# B&R Automation Studio project prak4
Automation Studio 4.5.2.102

## Configuration Config1

### Hardware
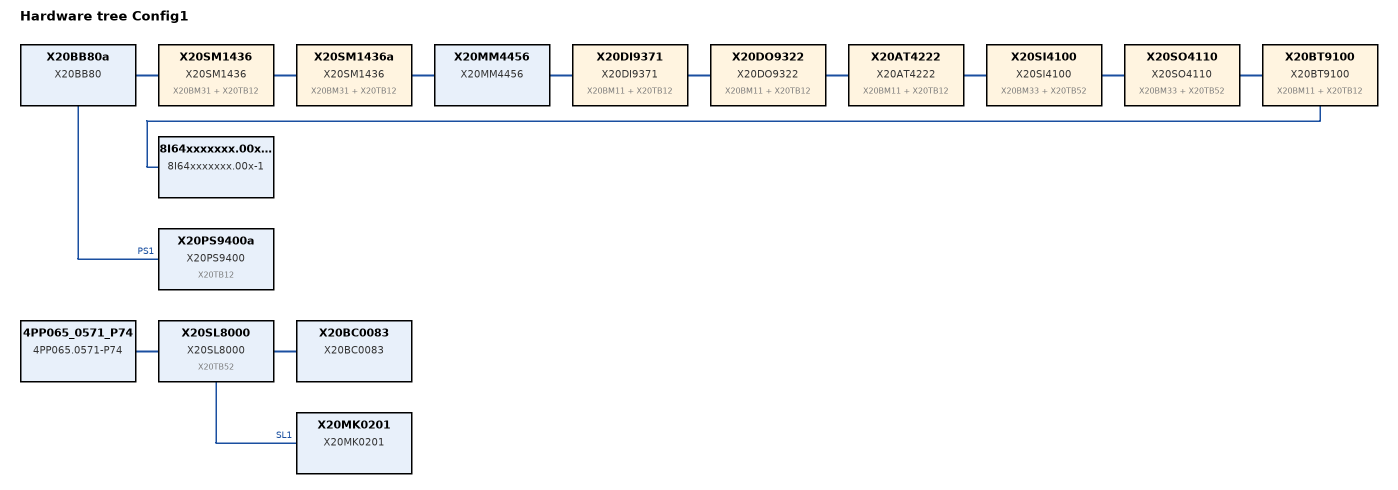
```
4PP065_0571_P74 : 4PP065.0571-P74 v1.1.2.0
  Connector IF5:
    ActivateDevice = 1
    Mode = Manual
    InternetAddress = 10.0.1.10
    SubnetMask = 255.255.255.0
  ConfigurationID = labBR
  TimerDeviceType = EPLX2X
  TimerDevice = 4PP065_0571_P74.IF4
  TaskClassIdleTime = 2000
  Cyclic1Duration = 2000
  Cyclic1Tolerance = 0
  Cyclic1Output = 1
  VcObjectName = Visu
8I64xxxxxxx.00x-1 : 8I64xxxxxxx.00x-1 v2.1.2.0  [X2X1 -> X20BT9100.X2X1 [Cable Type=X2XCable, Length=10, Version=1.0.0.2]]
  packedETAD = packed
  packedCMDD = packed
X20AT4222 : X20AT4222 v1.2.3.0  [SS1 -> X20TB12e.SS; SL -> X20BM11b.SL1]
X20BB80a : X20BB80 v1.0.2.0
X20BC0083 : X20BC0083 v2.9.0.0  [PLK1 -> X20SL8000.PLK2 [Cable Type=PowerlinkCable, Length=10, Version=1.0.0.2]; SL -> X20BB80a.SL1]
X20BM11 : X20BM11 v1.0.0.1  [X2X1 -> X20MM4456.X2X2]
X20BM11a : X20BM11 v1.0.0.1  [X2X1 -> X20BM11.X2X2]
X20BM11b : X20BM11 v1.0.0.1  [X2X1 -> X20BM11a.X2X2]
X20BM11c : X20BM11 v1.0.0.1  [X2X1 -> X20BM33a.X2X2]
X20BM31 : X20BM31 v1.0.0.1  [X2X1 -> X20BB80a.IF1]
X20BM31a : X20BM31 v1.0.0.1  [X2X1 -> X20BM31.X2X2]
X20BM33 : X20BM33 v1.0.0.4  [X2X1 -> X20BM11b.X2X2]
X20BM33a : X20BM33 v1.0.0.4  [X2X1 -> X20BM33.X2X2]
X20BT9100 : X20BT9100 v1.0.3.0  [SS1 -> X20TB12f.SS; SL -> X20BM11c.SL1]
X20DI9371 : X20DI9371 v1.0.2.0  [SS1 -> X20TB12c.SS; SL -> X20BM11.SL1]
X20DO9322 : X20DO9322 v1.0.3.0  [SS1 -> X20TB12d.SS; SL -> X20BM11a.SL1]
X20MK0201 : X20MK0201 v1.0.0.0  [SL -> X20SL8000.SL1]
X20MM4456 : X20MM4456 v1.1.5.0  [X2X1 -> X20BM31a.X2X2]
X20PS9400a : X20PS9400 v1.0.2.4  [SS1 -> X20TB12a.SS; PS -> X20BB80a.PS1]
X20SI4100 : X20SI4100 v1.10.1.1  [SS1 -> X20TB52a.SS; SL -> X20BM33.SL1]
X20SL8000 : X20SL8000 v1.6.5.1  [PLK1 -> 4PP065_0571_P74.IF4 [Cable Type=PowerlinkCable, Length=10, Version=1.0.0.2]; PLK2 -> X20BC0083.PLK1 [Cable Type=PowerlinkCable, Length=10, Version=1.0.0.2]; SS1 -> X20TB52.SS]
  SafeProject = SafeLOGIC-1
X20SM1436 : X20SM1436 v1.4.2.1  [SS1 -> X20TB12.SS; SL -> X20BM31.SL1]
X20SM1436a : X20SM1436 v1.4.2.1  [SS1 -> X20TB12b.SS; SL -> X20BM31a.SL1]
X20SO4110 : X20SO4110 v1.10.1.1  [SS1 -> X20TB52b.SS; SL -> X20BM33a.SL1]
  SafeModuleID = 3
X20TB12 : X20TB12 v1.0.0.0
X20TB12a : X20TB12 v1.0.0.0
X20TB12b : X20TB12 v1.0.0.0
X20TB12c : X20TB12 v1.0.0.0
X20TB12d : X20TB12 v1.0.0.0
X20TB12e : X20TB12 v1.0.0.0
X20TB12f : X20TB12 v1.0.0.0
X20TB52 : X20TB52 v1.0.0.1
X20TB52a : X20TB52 v1.0.0.1
X20TB52b : X20TB52 v1.0.0.1
```

### IoMap.iom - 4PP065_0571_P74/IoMap.iom
```iecst
VAR_CONFIG
	Cyclic#1.gAxis02_DrvIf.iLifeCnt AT %IB."8I64xxxxxxx.00x-1".SDC_LifeCnt;
	Cyclic#1.gAxis02_DrvIf.iDrvOK AT %IX."8I64xxxxxxx.00x-1".ETAD_Input_Bool_02;
	Cyclic#1.gAxis02_DrvIf.oSetTime AT %QW."8I64xxxxxxx.00x-1".SDC_SetTime;
	::Program:speed AT %QW."8I64xxxxxxx.00x-1".LFRD_Output;
	Cyclic#1.gAxis02_DiDoIf.iLifeCntDriveReady AT %IB."8I64xxxxxxx.00x-1".SDC_LifeCnt;
	Cyclic#1.gAxis02_DiDoIf.iLifeCntDriveEnable AT %IB."8I64xxxxxxx.00x-1".SDC_LifeCnt;
	Cyclic#1.gAxis02_DiDoIf.oDriveEnable AT %QX."8I64xxxxxxx.00x-1".CMDD_Output_Bool_00;
	Cyclic#1.gAxis02_ModuleOk AT %QX."8I64xxxxxxx.00x-1".CMDD_Output_Bool_01;
	Cyclic#1.gAxis02_ModuleOk AT %QX."8I64xxxxxxx.00x-1".CMDD_Output_Bool_02;
	Cyclic#1.gAxis02_ModuleOk AT %IX."8I64xxxxxxx.00x-1".ModuleOk;
	Cyclic#1.gAxis02_DiDoIf.oDriveEnable AT %QX."8I64xxxxxxx.00x-1".CMDD_Output_Bool_03;
	Cyclic#1.gAxis02_DiDoIf.iDriveReady AT %IX."8I64xxxxxxx.00x-1".ETAD_Input_Bool_02;
	EVIRD.STATE AT %IW."8I64xxxxxxx.00x-1".ETAD_Input;
	::EVIRD.COM AT %QW."8I64xxxxxxx.00x-1".CMDD_Output;
	::led1 AT %QX."X20DO9322".DigitalOutput02;
	::led2 AT %QX."X20DO9322".DigitalOutput03;
	::led3 AT %QX."X20DO9322".DigitalOutput04;
	::led4 AT %QX."X20DO9322".DigitalOutput05;
	::EVIRD.real_speed AT %IW."8I64xxxxxxx.00x-1".RFRD_Input;
END_VAR
```

### Acp10map.ncm - 4PP065_0571_P74/Motion/Acp10map.ncm
```
NcMapping (NcSwId=Acp10)
  NcObject X20SM1436_ncAXIS1 (ModuleId=X20SM1436, ModuleAddress=SDC_IF1.ST1, Type=ncAXIS, Channel=1, AcoposSimulation=Off, Disabled=TRUE, ModuleDisabled=FALSE)
  NcObject X20SM1436a_ncAXIS1 (ModuleId=X20SM1436a, ModuleAddress=SDC_IF1.ST2, Type=ncAXIS, Channel=1, AcoposSimulation=Off, Disabled=TRUE, ModuleDisabled=FALSE)
  NcObject gAxis02 (ModuleId=8I64xxxxxxx.00x-1, ModuleAddress=SDC_IF1.ST3, Type=ncAXIS, Channel=1, AcoposSimulation=Off, InitParameter=gAxis02i, AcoposParameter=gAxis02a, Disabled=FALSE, ModuleDisabled=FALSE)
```

## Logical view

Binary libraries used (declarations not repeated): operator, runtime, astime, AsIecCon, Acp10man, Acp10par, NcGlobal, Acp10sdc, AsBrStr, Acp10_MC, brsystem, sys_lib

### Global.var - Global variables
```iecst
VAR
	gAxis01 : ACP10AXIS_typ;
	gAxis01_HW : SdcHwCfg_typ := (0);
	gAxis01_DrvIf : SdcDrvIf16_typ := (0);
	gAxis01_DiDoIf : SdcDiDoIf_typ := (0);
	gAxis01_ModuleOk : BOOL := 0;
	gAxis02 : ACP10AXIS_typ;
	gAxis02_HW : SdcHwCfg_typ := (0);
	gAxis02_DrvIf : SdcDrvIf16_typ := (0);
	gAxis02_DiDoIf : SdcDiDoIf_typ := (0);
	gAxis02_ModuleOk : BOOL := 0;
	EVIRD : DRIVE;
	led1 : BOOL;
	led2 : BOOL;
	led3 : BOOL;
	led4 : BOOL;
END_VAR
```

### Package Logical/Libraries - Global libraries

- Visualisation Logical/Libraries/Visu (not shown)

### Program Logical/Program (ANSIC)

#### Variables.var
```iecst
VAR
	speed : INT;
END_VAR
```

#### Main.c
```c
#include <bur/plctypes.h>

#ifdef _DEFAULT_INCLUDES
	#include <AsDefault.h>
#endif

void _INIT ProgramInit(void)
{
	speed = 500;
	EVIRD.ENABLE=1;
}

void _CYCLIC ProgramCyclic(void)
{

	DRIVE(&EVIRD);
}

void _EXIT ProgramExit(void)
{

}
```

### Program Logical/ncsdcctrl (IEC)

#### ncsdcctrlCyclic.st
```iecst
PROGRAM _CYCLIC

(* ### BEGIN gAxis01 ### *)

(* life counter emulation of digital inputs *)
        gAxis01_DiDoIf.iLifeCntReference := gAxis01_DiDoIf.iLifeCntReference + 1;
        gAxis01_DiDoIf.iLifeCntNegHwEnd  := gAxis01_DiDoIf.iLifeCntNegHwEnd  + 1;
        gAxis01_DiDoIf.iLifeCntPosHwEnd  := gAxis01_DiDoIf.iLifeCntPosHwEnd  + 1;

(* ### END gAxis01 ### *)

(* ### BEGIN gAxis02 ### *)

(* life counter emulation of digital inputs *)
        gAxis02_DiDoIf.iLifeCntReference := gAxis02_DiDoIf.iLifeCntReference + 1;
        gAxis02_DiDoIf.iLifeCntNegHwEnd  := gAxis02_DiDoIf.iLifeCntNegHwEnd  + 1;
        gAxis02_DiDoIf.iLifeCntPosHwEnd  := gAxis02_DiDoIf.iLifeCntPosHwEnd  + 1;

(* ### END gAxis02 ### *)

END_PROGRAM
```

#### ncsdcctrlInit.st
```iecst
PROGRAM _INIT

(* ### BEGIN gAxis01 ### *)

(* initialize variables *)
        gAxis01_HW.DrvIf_Typ := ncSDC_DRVSERVO16;
        brsstrcpy(ADR(gAxis01_HW.DrvIf_Name[0]), ADR('gAxis01_DrvIf'));
        gAxis01_HW.DiDoIf_Typ := ncSDC_DIDO;
        brsstrcpy(ADR(gAxis01_HW.DiDoIf_Name[0]), ADR('gAxis01_DiDoIf'));

(* force variable offset generation *)
        gAxis01.size                      := gAxis01.size;
        gAxis01_DrvIf.iLifeCnt            := gAxis01_DrvIf.iLifeCnt;
        gAxis01_DiDoIf.iLifeCntDriveReady := gAxis01_DiDoIf.iLifeCntDriveReady;
        gAxis01_ModuleOk                  := gAxis01_ModuleOk;

(* assign your hardware inputs here*)

(*      gAxis01_DiDoIf.iPosHwEnd  := gAxis01_DiDoIf.iPosHwEnd;
        gAxis01_DiDoIf.iNegHwEnd  := gAxis01_DiDoIf.iNegHwEnd;
        gAxis01_DiDoIf.iReference := gAxis01_DiDoIf.iReference;
 *)

(* ### END gAxis01 ### *)

(* ### BEGIN gAxis02 ### *)

(* initialize variables *)
        gAxis02_HW.DrvIf_Typ := ncSDC_DRVSERVO16;
        brsstrcpy(ADR(gAxis02_HW.DrvIf_Name[0]), ADR('gAxis02_DrvIf'));
        gAxis02_HW.DiDoIf_Typ := ncSDC_DIDO;
        brsstrcpy(ADR(gAxis02_HW.DiDoIf_Name[0]), ADR('gAxis02_DiDoIf'));

(* force variable offset generation *)
        gAxis02.size                      := gAxis02.size;
        gAxis02_DrvIf.iLifeCnt            := gAxis02_DrvIf.iLifeCnt;
        gAxis02_DiDoIf.iLifeCntDriveReady := gAxis02_DiDoIf.iLifeCntDriveReady;
        gAxis02_ModuleOk                  := gAxis02_ModuleOk;

(* assign your hardware inputs here*)

(*      gAxis02_DiDoIf.iPosHwEnd  := gAxis02_DiDoIf.iPosHwEnd;
        gAxis02_DiDoIf.iNegHwEnd  := gAxis02_DiDoIf.iNegHwEnd;
        gAxis02_DiDoIf.iReference := gAxis02_DiDoIf.iReference;
 *)

(* ### END gAxis02 ### *)

END_PROGRAM
```

### Library Logical/Library (ANSIC)

#### Library.fun
```iecst
{REDUND_ERROR} FUNCTION_BLOCK DRIVE (*TODO: Add your comment here*) (*$GROUP=User,$CAT=User,$GROUPICON=User.png,$CATICON=User.png*)
	VAR_INPUT
		ENABLE : BOOL;
		STATE : UINT;
	END_VAR
	VAR_OUTPUT
		COM : UINT;
		real_speed : INT;
	END_VAR
END_FUNCTION_BLOCK
```

#### DRIVE.c
```c
#include <bur/plctypes.h>
#ifdef __cplusplus
	extern "C"
	{
#endif
	#include "Library.h"
#ifdef __cplusplus
	};
#endif
/* TODO: Add your comment here */
void DRIVE(struct DRIVE* inst)
{
	UINT mask=inst->STATE & 0x6f;
	if(!inst ->ENABLE)
	{
		inst ->COM = CMD_SHUTDOWN;
	}
	else
	{
		switch(mask)
		{
			case STATE_DISABLED:

				inst ->COM=CMD_SHUTDOWN;
				break;
			case STATE_READY:

				inst ->COM=CMD_ENABLED;
				break;

			case STATE_SWITCHED_ON:

				inst ->COM=CMD_SWITCHED_ON;
				break;
		}
	}
	/*TODO: Add your code here*/
}
```

### Program Logical/Program1 (ANSIC)

#### Variables.var
```iecst
VAR
	LED : ARRAY[0..3] OF BOOL;
END_VAR
```

#### Main.c
```c
#include <bur/plctypes.h>

#ifdef _DEFAULT_INCLUDES
	#include <AsDefault.h>
#endif

void _INIT ProgramInit(void)
{

}

void _CYCLIC ProgramCyclic(void)
{
	led1 = LED[0];
	led2 = LED[1];
	led3 = LED[2];
	led4 = LED[3];
}

void _EXIT ProgramExit(void)
{

}
```

Listed in the project but not available here: Logical/Global.typ, Logical/acp10etxen, Logical/gAxis01obj, Logical/gAxis02obj
